Fanuc KAREL source: kb00199.KL

-- PROVISIONAL review KL for V770-1; original PC SHA256 221bfdcaa916ab458b4e23b96f96f93e515cc0b5cef34d7a2ab51d7dcc7f34eb
-- Incomplete behavior may be omitted. Consult companion uncertainty JSON. Do not deploy.
PROGRAM KB00199
%NOLOCKGROUP
BEGIN
  -- UNRESOLVED_PC offsets 5-14; opcodes 3F,75
  -- UNRESOLVED_PC offsets 19-26; opcodes 9D,23
  -- UNRESOLVED_PC offsets 31-38; opcodes 9D,23
  -- UNRESOLVED_PC offsets 43-50; opcodes 9D,23
  -- UNRESOLVED_PC offsets 55-62; opcodes 9D,23
  -- UNRESOLVED_PC offsets 67-109; opcodes 27,22,22,2A,22,22,22,22,31
  -- UNRESOLVED_PC offsets 114-118; opcodes 7F
END KB00199
